FUNCTION_BLOCK fbValve_Solenoid
VAR_INPUT
	tInTimeout: TIME:=T#10S;		//The amount of time before an error condition triggers an error
	iInMode:	INT;		//system mode 1=Auto, 2=Manual, 10=Independent
	bInEstop:	BOOL;		//Emergency stop input 1=Estop
	bInSignalHome:	BOOL;	//Home position feedback
	bInSignalWork:	BOOL;	//Work position feedback
	bInEnable:		BOOL;	//Valve interlock. The valve is allowed to operate if this condition has been met
	bInCommandWork: BOOL;	//Move to work position in automatic mode
	bInResetError:	BOOL;	//If an error condition exists, the error must be fixed first, then set this bit high to reset the internal error
	bInSimulate:	BOOL;	//Enables software simulation of device.
END_VAR
VAR_OUTPUT
	bOutCommandHome: BOOL;	//Output for home position
	bOutCommandWork: BOOL;	//Output for work position
	bOutActiveHome: BOOL;	//Valve is actively in home position
	bOutActiveWork: BOOL;	//Valve is actively in work position
	bOutAuto: BOOL;			//This output indicates whether the block is in auto mode
	bOutError: BOOL;		//This output indicates whether there's an error condition in the cylinder
	ERROR_Valve:stError_Valve;
END_VAR

VAR_IN_OUT
	HMI_ValveControl:stHMI_ValveControl;
END_VAR

VAR
	tonTimeOut:TON;
	iErrorCode:INT;
	bNewMode:BOOL;	 (*new mode selected*)
	bAutoMode:BOOL;	 (*Automode active*)
	bManualMode:BOOL; (*Manual Mode active*)
	iLastMode:INT;	(*last mode code*)
	bEnableHome:BOOL;	 (*home position enabled*)
	bEnableWork:BOOL;	 (*work position enabled*)
	bPB_Home:BOOL;		 (*PB Move to home in manual mode*)
	bPB_Work:BOOL;		 (*PB Move to work in manual mode*)
	bPB_ResetError:BOOL; (*PB Reset error*)
	bReset: BOOL;
	handleHMIBit1,handleHMIBit2,handleHMIBit3:fbHMIBit;
END_VAR



(*****************************INPUTS*************************************************)
(*Read HMI input button*)

handleHMIBit1(bInToggle:=1 , bHMI:=HMI_ValveControl.bPB_Home , bPLC:=bPB_Home );  
handleHMIBit2(bInToggle:=1 , bHMI:=HMI_ValveControl.bPB_Work , bPLC:=bPB_Work ); 
handleHMIBit2(bInToggle:=1 , bHMI:=HMI_ValveControl.bPB_ResetError , bPLC:=bPB_ResetError ); 


(*update the signal home bit*)
HMI_ValveControl.bSignalHome:=bInSignalHome;

(*update the signal work bit*)
HMI_ValveControl.bSignalWork:=bInSignalWork;

(**************************CONTROL LOGIC************************************************)
(*Clear all errors*)
IF (bInResetError OR bPB_ResetError) AND HMI_ValveControl.bPB_ResetError THEN
	bReset:=1;
ELSE 
	bReset:=0;
END_IF


(*override HMI mode if not in Independant mode*)
IF iInMode<>10 THEN
	HMI_ValveControl.iMode:=iInMode;
END_IF

(*detect change in mode*)
bNewMode:=HMI_ValveControl.iMode<>iLastMode;

(*keep track of last mode*)
iLastMode:=HMI_ValveControl.iMode;

(*Determine if auto or manual mode Active*)
bManualMode:=NOT(bInEstop) AND NOT(bNewMode) AND (HMI_ValveControl.iMode=2);
bAutoMode:=NOT(bInEstop) AND NOT(bNewMode) AND (HMI_ValveControl.iMode=1);

(*Enable home and work positions*)
bEnableWork:=bEnableHome:= NOT(HMI_ValveControl.bError) AND (bManualMode OR bAutoMode);

HMI_ValveControl.bPBEN_Home:=HMI_ValveControl.bPBEN_Work:=bManualMode AND NOT(HMI_ValveControl.bError);

(*enable error reset button if error present*)
HMI_ValveControl.bPBEN_ResetError:=HMI_ValveControl.bPB_ResetError;

(*Command Home position*)
IF (bManualMode AND bPB_Home AND  NOT(bPB_Work) AND HMI_ValveControl.bPBEN_Home) OR
	(bAutoMode AND NOT(bInCommandWork) AND bEnableHome) THEN
	HMI_ValveControl.bHomeOn:=1;
	HMI_ValveControl.bWorkOn:=0;
END_IF

(*command work position*)
IF (bManualMode AND bPB_Work AND  NOT(bPB_Home) AND HMI_ValveControl.bPBEN_Work) OR
	(bAutoMode AND bInCommandWork AND bEnableWork) THEN
	HMI_ValveControl.bWorkOn:=1;
	HMI_ValveControl.bHomeOn:=0;
END_IF

(*reset work if not enabled*)
IF bAutoMode AND NOT(bEnableWork) THEN
	HMI_ValveControl.bWorkOn:=0;
END_IF

(*reset home if not enabled*)
IF bAutoMode AND NOT(bEnableHome) THEN
	HMI_ValveControl.bHomeOn:=0;
END_IF

(*if Not in auto or manual reset both*)
IF NOT(bAutoMode OR bManualMode) THEN
	HMI_ValveControl.bHomeOn:=0;
	HMI_ValveControl.bWorkOn:=0;
END_IF

(************************************ERRORS*************************************************************)
(*set timeout errors*)
tonTimeOut(IN:=HMI_ValveControl.bHomeOn OR HMI_ValveControl.bWorkOn , PT:= , Q=> , ET=> );

(*Error: Work Feedback not active*)
ERROR_Valve.NoWorkFeedback:=NOT(bInEstop) AND tonTimeOut.Q AND HMI_ValveControl.bWorkOn AND NOT(HMI_ValveControl.bSignalWork);

(*Error: Home feedback not active*)
ERROR_Valve.NoHomeFeedback:=NOT(bInEstop) AND tonTimeOut.Q AND HMI_ValveControl.bHomeOn AND NOT(HMI_ValveControl.bSignalHome);

(*Error: Home position still active*)
ERROR_Valve.HomeFeedbackStillActive:=NOT(bInEstop) AND tonTimeOut.Q AND HMI_ValveControl.bWorkOn AND HMI_ValveControl.bSignalHome;

(*Error: Work position still active*)
ERROR_Valve.WorkFeedbackStillActive:=NOT(bInEstop) AND tonTimeOut.Q AND HMI_ValveControl.bHomeOn AND HMI_ValveControl.bSignalWork;

HMI_ValveControl.iErrorCode.0:=ERROR_Valve.NoWorkFeedback;
HMI_ValveControl.iErrorCode.1:=ERROR_Valve.NoHomeFeedback;
HMI_ValveControl.iErrorCode.2:=ERROR_Valve.HomeFeedbackStillActive;
HMI_ValveControl.iErrorCode.3:=ERROR_Valve.WorkFeedbackStillActive;

HMI_ValveControl.bError:=HMI_ValveControl.iErrorCode<>0;

(*Interlock*)
HMI_ValveControl.bInterlock:=bInEnable;

(************************************OUTPUTS**********************************************************************************)
(*Output Home*)
bOutCommandHome:=HMI_ValveControl.bHomeOn;

(*Output Work*)
bOutCommandWork:=HMI_ValveControl.bWorkOn;

(*Output Auto*)
bOutAuto:=(HMI_ValveControl.iMode=1);

(*Output error*)
bOutError:=HMI_ValveControl.bError;

END_FUNCTION_BLOCK

(* stored: Version 1.1.0.1, ProductVersion 3.1.4024.11
   POU fbValve_Solenoid: Id {4590884d-7356-4537-bc1e-3a60dfcf47a8}, SpecialFunc None *)
